PROGRAM MAIN
VAR
	PlayInTraffic:BOOL:=FALSE;
END_VAR

// <- this is how you comment out lines, anything after the // will not be part of the program 
//this is how you can leave notes for future developers or if code isn't working right you can remove it temporarily to test things without deleting it  
Ladder(); //This calls the ladder logic example
StructuredText(); //This calls the structured text example

IF PlayInTraffic THEN
	TrafficManager();
END_IF

END_PROGRAM

(* stored: Version 1.1.0.1, ProductVersion 3.1.4024.11
   POU MAIN: Id {b666fc23-fe06-4f53-8f48-ffbc045e9268}, SpecialFunc None *)
